TYPE SafetyConfig :
STRUCT
	///Some configuration values of the Dome Access
	domeAccess: SafetyDomeAccessConfig;
END_STRUCT
END_TYPE

(* stored: Version 1.1.0.1, ProductVersion 3.1.4019.2
   DUT SafetyConfig: Id {1dea4806-1f24-43c6-a79d-d51a9fcb0a23} *)
